// TIA Portal V19 export
FUNCTION "FC_DB_COPY" : Void   // FC3, STL
TITLE = Blocktransfer
{ S7_Optimized_Access := 'FALSE' }
AUTHOR : MS
// Kopiert Datenblöcke von Quell- zu Ziel-DB und löscht(bei CLR_ALT_DB) 
// anschließend eingetragenen Bereich im Quell-Db
// stored: AutoNumber false
   VAR_INPUT
      CLR_ALT_DB : Bool;   // NACH DEM KOPIEREN WIRD DER URSPRUNG-DB GELÖSCHT
      ALT_DB : Int;   // URSPRUNG DB
      NEU_DB : Int;   // ZIEL DB
      COPY_START : Int;   // ADRESSE DES WORTES, WELCHES ALS ERSTES KOPIERT WIRD
      COPY_ENDE : Int;   // ADRESSE DES WORTES, WELCHES ALS ERSTES NICHT MEHR KOPIERT WIRD
      ZIEL_START : Int;   // STARTADRESSE DATENBEREICH ZIEL
      CLR_START : Int;   // ADRESSE DES WORTES, WELCHES ALS ERSTES GELÖSCHT WIRD
      CLR_ENDE : Int;   // ADRESSE DES WORTES, WELCHES ALS ERSTES NICHT MEHR GELÖSCHT WIRD
   END_VAR
   VAR_IN_OUT
      START : Bool;   // DURCHLAUFMERKER/OK-SIGNAL
   END_VAR
   VAR_TEMP
      ZAEHLER1 : Int;   // ZAEHLVARIABLE QUELLE
      ZAEHLER2 : Int;   // ZAEHLVARIABLE ZIEL
      Alt_DB1 : Word;
      Neu_DB1 : Word;
   END_VAR
BEGIN

NETWORK
TITLE = Copy
// DATENBEREICH KOPIEREN
      L     #ALT_DB;
      T     #Alt_DB1;
      OPN   DI [#Alt_DB1];
      L     #NEU_DB;
      T     #Neu_DB1;
      OPN   DB [#Neu_DB1];
      AN    #START;
      BEC;
      L     #COPY_START;
      T     #ZAEHLER1;
      L     #ZIEL_START;
      T     #ZAEHLER2;
COPY: L     #ZAEHLER1;
      SLD   3;
      LAR1;
      L     #ZAEHLER2;
      SLD   3;
      LAR2;
      L     DIW [AR1, P#0.0];
      T     DBW [AR2, P#0.0];
      L     #ZAEHLER2;
      L     2;
      +D;
      T     #ZAEHLER2;
      L     #ZAEHLER1;
      L     2;
      +D;
      T     #ZAEHLER1;
      L     #COPY_ENDE;
      <I;
      JC    COPY;

NETWORK
TITLE = Delete
// DATENBEREICH DER QUELLE MIT "0" FÜLLEN
      AN    #CLR_ALT_DB;
      JC    AUS;
      L     #CLR_START;  //STARTADRESSE WORT LÖSCHEN
      T     #ZAEHLER1;
DEL:  L     #ZAEHLER1;
      SLD   3;
      LAR1;
      L     0;
      T     DIW [AR1, P#0.0];
      L     #ZAEHLER1;
      L     2;
      +D;
      T     #ZAEHLER1;
      L     #CLR_ENDE;  //ENDADRESSE WORT LÖSCHEN
      <I;
      JC    DEL;

NETWORK
TITLE = Ready
// ENDE /FERTIGMELDUNG
AUS:  CLR;
      =     #START;
      BE;
END_FUNCTION
